INTERFACE I_MqttDeviceDiscoveryProvider

METHOD GetMqttDeviceDiscovery : I_MqttDeviceDiscovery
VAR_INPUT
END_VAR
END_METHOD

END_INTERFACE

(* stored: Version 1.1.0.1, ProductVersion 3.1.4024.5
   Itf I_MqttDeviceDiscoveryProvider: Id {f3644253-7c52-45bf-a602-bd3dbc5088a5}
   Method GetMqttDeviceDiscovery: Id {58f72f22-8a5a-4387-b568-4c9c2ab69278} *)
